# EPICS autosave request: LabJackApp/Db/LabJack_ao_settings.req
$(P)Ao$(N).LOPR
$(P)Ao$(N).HOPR
$(P)Ao$(N).EGUF
$(P)Ao$(N).EGUL
$(P)Ao$(N).PREC
$(P)Ao$(N).DESC
$(P)Ao$(N)TweakVal
